{attribute addProperty BoxType "EP1816-0008-0016"}
{attribute addProperty Id "DO_Inputs_ChannelAT %I*ARRAY[0..1] OF DO_Inputs_Channel_9F71B9E2144180WcStateAT %I*WcState_F855686C1620InfoDataAT %I*InfoData_BC63D37F80100"}
{attribute addProperty CRC "2234885487"}
{attribute addProperty SizeInBites "240"}
{attribute addProperty SizeInBytes "30"}
TYPE EP1816_D737114C :
STRUCT
	{attribute addProperty Name "DO_Inputs_Channel"}
	DO_Inputs_Channel : ARRAY[0..1] OF DO_Inputs_Channel_9F71B9E2;
	{attribute addProperty Name "WcState"}
	WcState : WcState_F855686C;
	{attribute addProperty Name "InfoData"}
	InfoData : InfoData_BC63D37F;
END_STRUCT
END_TYPE

(* stored: Version 1.2.0.0, ProductVersion 3.1.4024.9
   DUT EP1816_D737114C: Id {da529c24-3470-4910-8495-17491313d27e} *)
